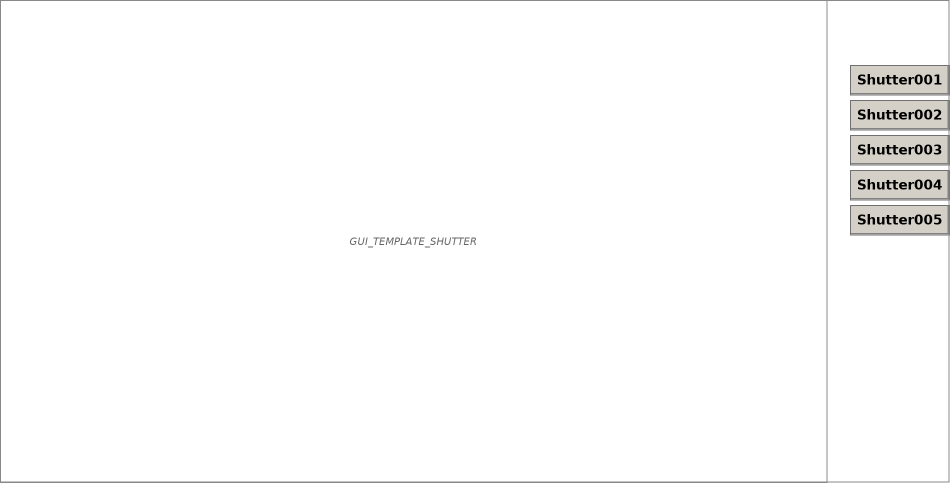
VISUALIZATION GUI_All  // 950x483
    Frame (0,0 827x483)
        shows GUI_TEMPLATE_SHUTTER(m_Instance := MAIN.ptrGUI_Shutters[MAIN.nPtrIndex_Shutters]^)
    Button (850,65 100x30), "Shutter001"
        OnMouseClick: execute { MAIN.nPtrIndex_Shutters:=1; }
    Button (850,100 100x30), "Shutter002"
        OnMouseClick: execute { MAIN.nPtrIndex_Shutters:=2; }
    Button (850,135 100x30), "Shutter003"
        OnMouseClick: execute { MAIN.nPtrIndex_Shutters:=3; }
    Button (850,170 100x30), "Shutter004"
        OnMouseClick: execute { MAIN.nPtrIndex_Shutters:=4; }
    Button (850,205 100x30), "Shutter005"
        OnMouseClick: execute { MAIN.nPtrIndex_Shutters:=5; }
END_VISUALIZATION

(* stored: Version 1.1.0.1, ProductVersion 3.1.4024.3
   Visu GUI_All: Id {ba6b4829-cfe8-4c1b-80a7-d8c3b6d4dc60} *)
